// TIA Portal V18 export
ORGANIZATION_BLOCK "Main"   // OB1, LAD, ProgramCycle
TITLE = "Main Program Sweep (Cycle)"
{ S7_Optimized_Access := 'TRUE' }
VERSION : 0.1
// stored: AutoNumber true, IsIECCheckEnabled false, SetENOAutomatically false
   VAR_INPUT
      Initial_Call : Bool;   // Initial call of this OB
      Remanence : Bool;   // =True, if remanent data are available
   END_VAR
BEGIN

REGION Network 1: Flow measurement
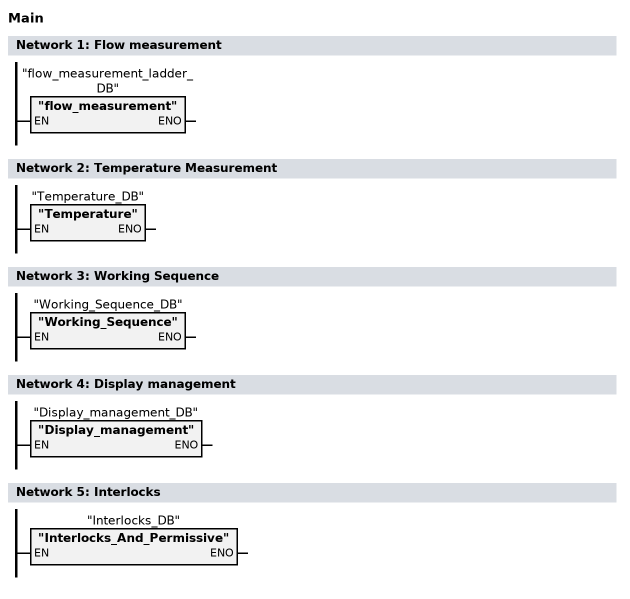
   RUNG wire#powerrail
      "flow_measurement_ladder_DB"()
   END_RUNG
   // the same network as SCL:
   "flow_measurement_ladder_DB"();   // "flow_measurement"
END_REGION

REGION Network 2: Temperature Measurement
   RUNG wire#powerrail
      "Temperature_DB"()
   END_RUNG
   // the same network as SCL:
   "Temperature_DB"();   // "Temperature"
END_REGION

REGION Network 3: Working Sequence
   RUNG wire#powerrail
      "Working_Sequence_DB"()
   END_RUNG
   // the same network as SCL:
   "Working_Sequence_DB"();   // "Working_Sequence"
END_REGION

REGION Network 4: Display management
   RUNG wire#powerrail
      "Display_management_DB"()
   END_RUNG
   // the same network as SCL:
   "Display_management_DB"();   // "Display_management"
END_REGION

REGION Network 5: Interlocks
   RUNG wire#powerrail
      "Interlocks_DB"()
   END_RUNG
   // the same network as SCL:
   "Interlocks_DB"();   // "Interlocks_And_Permissive"
END_REGION

REGION Network 6 (SCL): Emergency redundant signals
   // This is final command to ESD and the pump as a redundant command
   "To_contactor" := "To_contactor" AND "Var".emergency_state;
   "ESD_solenoid_valve" := "ESD_solenoid_valve" AND "Var".emergency_state;
END_REGION
END_ORGANIZATION_BLOCK
